PROGRAM MAIN_loggning
VAR
	fbIoT : FB_IoT_Publisher;
END_VAR

(*Energimatare Schneider*)
IF GVL_Fastighet.CSVEnergyMeter THEN
	iEM3255_Logg();
END_IF

(*Cluster Control*)
IF GVL_Fastighet.CSVClusterCtrl THEN
	Cluster_Logg();
	Cluster_Logg_2();
	Cluster_Logg_3();
	Cluster_Sensor_Logg();
END_IF

(*Vaderstation*)
IF GVL_Fastighet.CSVWXT530 THEN
	WXT530_Logg();
END_IF

(*Temperaturgivare*)
IF GVL_Fastighet.CSVTempProbes THEN
	Temp_Logg();
END_IF
//SOLINSTRÅLNINGS MÄTARE
IF GVL_Fastighet.CSVSR05 THEN
	SR05_Logg();
END_IF

//IoT
fbIoT();

END_PROGRAM

(* stored: Version 1.1.0.1, ProductVersion 3.1.4022.7
   POU MAIN_loggning: Id {72947dd7-2af7-418e-a96e-fb391ad9d335}, SpecialFunc None *)
